// TIA Portal V20 export
VAR_GLOBAL   // PLC tag table "Digital_Inputs"
   DI_FreeI0_0 AT %I0.0 : Bool;
   DI_X_AxisBrakePressCtrl AT %I0.1 : Bool;
   DI_Y_AxisBrakePressCtrl AT %I0.2 : Bool;
   DI_BreakerCtrl AT %I0.3 : Bool;
   DI_CabinetTemperatureCtrl AT %I0.4 : Bool;
   DI_UPS_PowerFailure AT %I0.5 : Bool;
   DI_AirPressureCtrl AT %I0.6 : Bool;
   DI_ShutterClosed AT %I0.7 : Bool;
   DI_AirDryerOK AT %I1.0 : Bool;
   DI_UPS_BatteryOK AT %I1.1 : Bool;
   DI_FrontDoorClosed AT %I1.2 : Bool;
   DI_InfeedReadyOK_Start AT %I1.3 : Bool;
   DI_CoolingOK AT %I1.4 : Bool;
   DI_FreeI1_5 AT %I1.5 : Bool;
   DI_PowerReady AT %I1.6 : Bool;
   DI_AlarmI2T AT %I1.7 : Bool;
   DI_HeadLaserBusy AT %I2.0 : Bool;
   DI_HeadLaserBreaker AT %I2.1 : Bool;
   DI_FrontDoorLocked AT %I2.2 : Bool;
   DI_UPS_CommonAlarm AT %I2.3 : Bool;
   DI_UPS_BatteryLow AT %I2.4 : Bool;
   DI_FreeI2_5 AT %I2.5 : Bool;
   DI_HeadChillerHighPressure AT %I2.6 : Bool;
   DI_HeadChillerWaterTemperature AT %I2.7 : Bool;
   DI_HeadChillerFlow AT %I3.0 : Bool;
   DI_HeadChillerCollectivFault AT %I3.1 : Bool;
   DI_HeadChillerWaterLevel AT %I3.2 : Bool;
   DI_UPSByPassActive AT %I3.3 : Bool;
   DI_HeadChillerAmbiantTemperature AT %I3.4 : Bool;
   DI_FreeI3_5 AT %I3.5 : Bool;
   DI_FreeI3_6 AT %I3.6 : Bool;
   DI_FreeI3_7 AT %I3.7 : Bool;
   DI_LoadClampOpened AT %I4.0 : Bool;
   DI_LoadClampNotClosedWithPart AT %I4.1 : Bool;
   DI_UnloadClampOpened AT %I4.2 : Bool;
   DI_UPS_Fault AT %I4.3 : Bool;
   DI_InternalGateLocked AT %I4.4 : Bool;
   DI_ExternalGateLocked AT %I4.5 : Bool;
   DI_InverterActive AT %I4.6 : Bool;
   DI_UnloadClampNotClosedWithPart AT %I4.7 : Bool;
   DI_FreeI5_0 AT %I5.0 : Bool;
   DI_FreeI5_1 AT %I5.1 : Bool;
   DI_InternalGateOpened AT %I5.2 : Bool;
   DI_ExternalGateOpened AT %I5.3 : Bool;
   DI_PowerMeterBackCtrl AT %I5.4 : Bool;
   DI_PowerMeterFrontCtrl AT %I5.5 : Bool;
   DI_FreeI5_6 AT %I5.6 : Bool;
   DI_FreeI5_7 AT %I5.7 : Bool;
   DI_HeadChillerCutOff AT %I6.0 : Bool;
   DI_HeadChillerTemperature AT %I6.1 : Bool;
   DI_FreeI6_2 AT %I6.2 : Bool;
   DI_FreeI6_3 AT %I6.3 : Bool;
   DI_ClampingOpenCtrl AT %I6.4 : Bool;
   DI_B_AxisBrakeReleasedCtrl AT %I6.5 : Bool;
   "DI_FreeI6.6" AT %I6.6 : Bool;
   DI_B_AxisReferencePoint AT %I6.7 : Bool;
   DI_SourceChillerHighPressure AT %I7.0 : Bool;
   DI_SourceChillerWaterTemperature AT %I7.1 : Bool;
   DI_SourceChillerFlow AT %I7.2 : Bool;
   DI_SourceChillerCollectivFault AT %I7.3 : Bool;
   DI_SourceChillerWaterLevel AT %I7.4 : Bool;
   DI_SourceChillerAmbiantTemperature AT %I7.5 : Bool;
   DI_SourceChillerCutOff AT %I7.6 : Bool;
   DI_SourceChillerTemperature AT %I7.7 : Bool;
END_VAR
